(* PLC project LD_self-hold.project, CODESYS CODESYS V3.5 SP15 Patch 3 *)
(* stored: creationDateTime 2020-12-19T08:50:39.1116389, modificationDateTime 2020-12-19T08:47:31.8389292 *)

PROGRAM POU
  VAR_INPUT
    X1 : BOOL;
    X2 : BOOL;
  END_VAR
  VAR_OUTPUT
    Y1 : BOOL;
  END_VAR

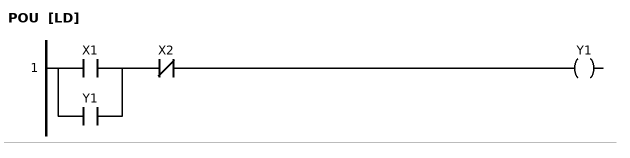
(* LD diagram, written out as Structured Text *)

Y1 := (X1 OR Y1) AND NOT X2;
END_PROGRAM
